// TIA Portal V20 export
DATA_BLOCK "Date and Time"   // DB3
{ S7_Optimized_Access := 'FALSE' }
AUTHOR : L.P.
// stored: AutoNumber false
   VAR RETAIN
      MEM : Struct
         "set by host" : Bool;
         "HM imp set by host" : Bool;
         "HM imp set by HMI" : Bool := false;
         "4" : Bool := false;
         "5" : Bool := false;
         "6" : Bool := false;
         "7" : Bool := false;
         "8" : Bool := false;
         "9" : Bool := false;
         "10" : Bool := false;
      END_STRUCT;
      "STEP" : Struct
         "0" : Bool;
         "1" : Bool;
         "2" : Bool;
         "3" : Bool;
         "4" : Bool;
         "5" : Bool;
         "6" : Bool;
         "7" : Bool;
         "8" : Bool;
         "9" : Bool;
         "10" : Bool;
      END_STRUCT;
      T : Struct
         "1" { S7_SetPoint := 'True'} : IEC_TIMER;
         "2" { S7_SetPoint := 'True'} : IEC_TIMER;
         "3" { S7_SetPoint := 'True'} : IEC_TIMER;
         "4" { S7_SetPoint := 'True'} : IEC_TIMER;
         "5" { S7_SetPoint := 'True'} : IEC_TIMER;
         "6" { S7_SetPoint := 'True'} : IEC_TIMER;
         "7" { S7_SetPoint := 'True'} : IEC_TIMER;
         "8" { S7_SetPoint := 'True'} : IEC_TIMER;
         "9" { S7_SetPoint := 'True'} : IEC_TIMER;
         "10" { S7_SetPoint := 'True'} : IEC_TIMER;
      END_STRUCT;
      C : Struct
         "1" { S7_SetPoint := 'True'} : IEC_COUNTER;
         "2" { S7_SetPoint := 'True'} : IEC_COUNTER;
         "3" { S7_SetPoint := 'True'} : IEC_COUNTER;
         "4" { S7_SetPoint := 'True'} : IEC_COUNTER;
         "5" { S7_SetPoint := 'True'} : IEC_COUNTER;
         "6" { S7_SetPoint := 'True'} : IEC_COUNTER;
         "7" { S7_SetPoint := 'True'} : IEC_COUNTER;
         "8" { S7_SetPoint := 'True'} : IEC_COUNTER;
         "9" { S7_SetPoint := 'True'} : IEC_COUNTER;
         "10" { S7_SetPoint := 'True'} : IEC_COUNTER;
      END_STRUCT;
      DATA : Struct
         "in date OP" : Date;
         "in time OP" : Time_Of_Day;
         "in date and time" : DTL;
         "out date and time" : DTL;
         year : UInt;
         month : USInt;
         day : USInt;
         hour : USInt;
         minute : USInt;
         second : USInt;
         millisecond : UInt;
         "day of week" : USInt;
         "day of year" : Int;
         "is Time Master" : Bool := true;
      END_STRUCT;
      BUTTON : Struct
         "set date and time" : Bool;
         "2" : Bool;
         "3" : Bool;
         "4" : Bool;
         "5" : Bool;
         "6" : Bool;
         "7" : Bool;
         "8" : Bool;
         "9" : Bool;
         "10" : Bool;
         "11" : Bool := false;
         "12" : Bool := false;
         "13" : Bool := false;
         "14" : Bool := false;
         "15" : Bool := false;
         "16" : Bool := false;
         "17" : Bool := false;
         "18" : Bool := false;
         "19" : Bool := false;
         "20" : Bool := false;
         "21" : Bool := false;
         "22" : Bool := false;
         "23" : Bool := false;
         "24" : Bool := false;
         "25" : Bool := false;
         "26" : Bool := false;
         "27" : Bool := false;
         "28" : Bool := false;
         "29" : Bool := false;
         "30" : Bool := false;
         "31" : Bool := false;
         "32" : Bool := false;
         "33" : Bool := false;
         "34" : Bool := false;
         "35" : Bool := false;
         "36" : Bool := false;
         "37" : Bool := false;
         "38" : Bool := false;
         "39" : Bool := false;
         "40" : Bool := false;
      END_STRUCT;
   END_VAR
BEGIN
END_DATA_BLOCK
